TYPE ST_System_Bel_Parameter :
STRUCT
	AutoQuittierung				: BOOL ;
	Zeit_Vorl					: DINT ; (* milisecs *)
	Zeit_Nachl					: DINT ; (* milisecs *)
	Stellwert_Leistung_max		: REAL ;
	Stellwert_Leistung_min		: REAL ;




	Nachtabsenkung_Uhrzeit_Stunde_Start			: REAL;	(* in 0-24h ggf. am Vortag *)
	Nachtabsenkung_Uhrzeit_Stunde_Ende			: REAL;	(* in 0-24h *)


END_STRUCT
END_TYPE

(* stored: Version 1.1.0.1, ProductVersion 3.1.4024.10
   DUT ST_System_Bel_Parameter: Id {1d16c3e4-5c59-4af6-a2e2-ee4354ef6d08} *)
